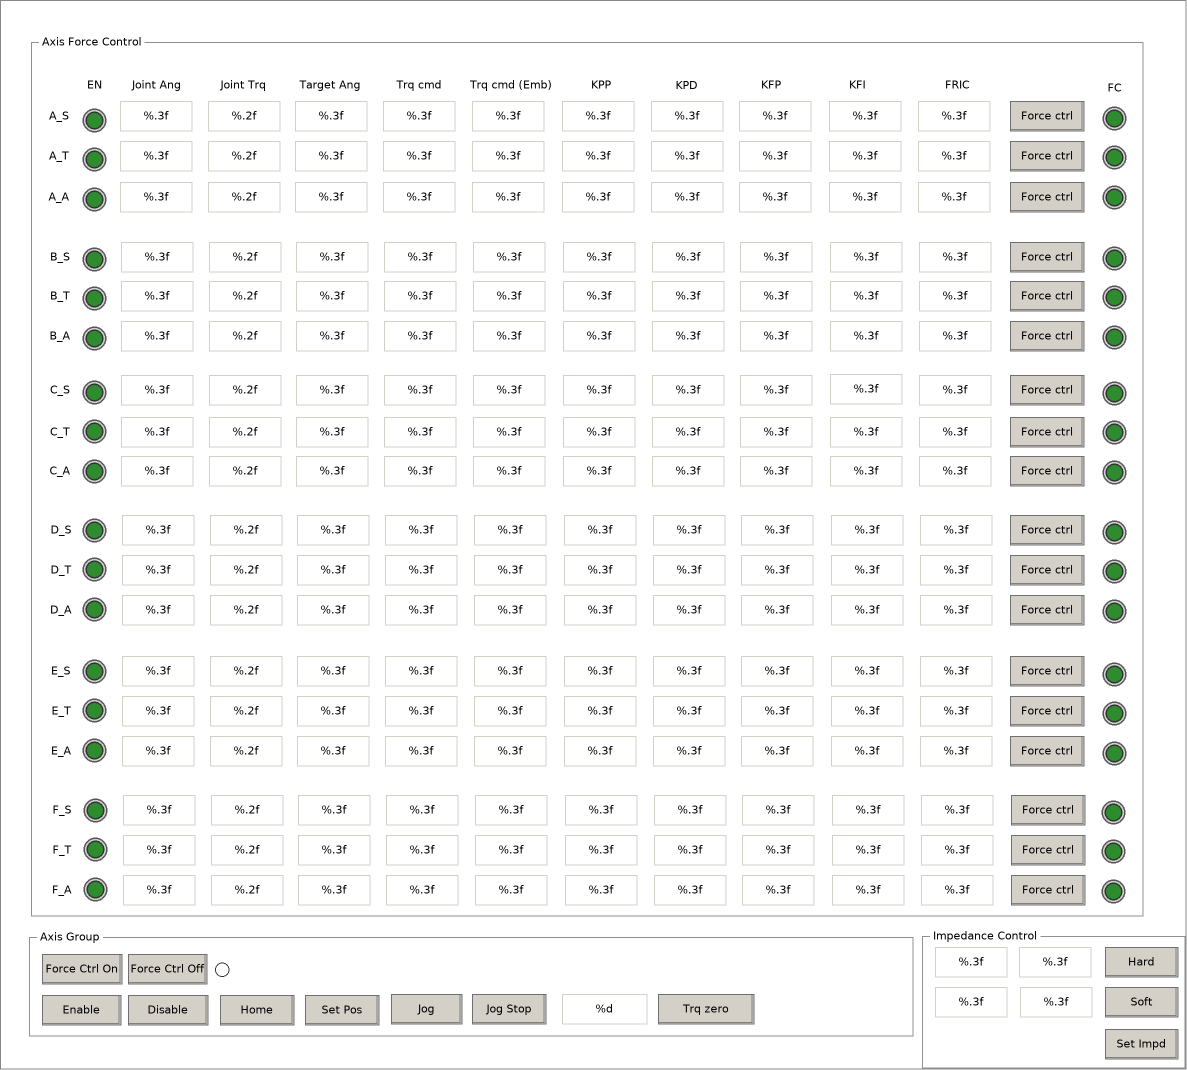
VISUALIZATION ForceControl  // 1187x1070
    GroupBox (31,34 1112x882), "Axis Force Control"
        Label (90,36 71x30), "Joint Ang"
        Label (179,36 67x30), "Joint Trq"
        Label (263,36 72x30), "Target Ang"
        Label (353,36 70x30), "Trq cmd"
        Label (433,36 94x30), "Trq cmd (Emb)"
        Textfield (89,67 72x30), "%.3f", text variable: GVL.motorDrive[0].motorAngle
        Label (545,39 50x24), "KPP"
        Label (632,36 47x31), "KPD"
        Label (800,36 53x30), "KFI"
        Label (714,36 52x30), "KFP"
        Label (900,36 53x30), "FRIC"
        Label (7,72 42x20), "A_S"
        Label (7,112 42x20), "A_T"
        Label (7,153 42x20), "A_A"
        Label (8,213 42x20), "B_S"
        Label (8,252 42x20), "B_T"
        Label (8,292 42x20), "B_A"
        Label (8,346 42x20), "C_S"
        Label (8,388 42x20), "C_T"
        Label (8,427 42x20), "C_A"
        Label (9,486 42x20), "D_S"
        Label (9,526 42x20), "D_T"
        Label (9,566 42x20), "D_A"
        Textfield (89,107 72x30), "%.3f", text variable: GVL.motorDrive[1].motorAngle
        Textfield (89,148 72x30), "%.3f", text variable: GVL.motorDrive[2].motorAngle
        Textfield (90,208 72x30), "%.3f", text variable: GVL.motorDrive[3].motorAngle
        Textfield (90,247 72x30), "%.3f", text variable: GVL.motorDrive[4].motorAngle
        Textfield (90,287 72x30), "%.3f", text variable: GVL.motorDrive[5].motorAngle
        Textfield (91,481 72x30), "%.3f", text variable: GVL.motorDrive[9].motorAngle
        Textfield (177,67 72x30), "%.2f", text variable: GVL.motorDrive[0].trqCalibrated
        Textfield (264,67 72x30), "%.3f", text variable: GVL.motorDrive[0].tgtAngle
            OnMouseClick: write the text variable via Default
        Textfield (352,67 72x30), "%.3f", text variable: GVL.motorDrive[0].trqOutput
        Button (979,67 74x30), "Force ctrl"
            toggle GVL.axisForceCtrlButton[0]
        Button (979,107 74x30), "Force ctrl"
            toggle GVL.axisForceCtrlButton[1]
        Button (979,148 74x30), "Force ctrl"
            toggle GVL.axisForceCtrlButton[2]
        Button (979,208 74x30), "Force ctrl"
            toggle GVL.axisForceCtrlButton[3]
        Button (979,247 74x30), "Force ctrl"
            toggle GVL.axisForceCtrlButton[4]
        Button (979,287 74x30), "Force ctrl"
            toggle GVL.axisForceCtrlButton[5]
        Button (979,341 74x30), "Force ctrl"
            toggle GVL.axisForceCtrlButton[6]
        Button (979,383 74x30), "Force ctrl"
            toggle GVL.axisForceCtrlButton[7]
        Button (979,422 74x30), "Force ctrl"
            toggle GVL.axisForceCtrlButton[8]
        Button (979,481 74x30), "Force ctrl"
            toggle GVL.axisForceCtrlButton[9]
        Button (979,521 74x30), "Force ctrl"
            toggle GVL.axisForceCtrlButton[10]
        Button (979,561 74x30), "Force ctrl"
            toggle GVL.axisForceCtrlButton[11]
        Textfield (620,67 72x30), "%.3f", text variable: GVL.motorDrive[0].bVirtual
            OnMouseClick: write the text variable via Default
        Textfield (708,67 72x30), "%.3f", text variable: GVL.motorDrive[0].kpTrqLoop
            OnMouseClick: write the text variable via Default
        Textfield (798,67 72x30), "%.3f", text variable: GVL.motorDrive[0].kiTrqLoop
            OnMouseClick: write the text variable via Default
        Textfield (887,67 72x30), "%.3f", text variable: GVL.motorDrive[0].reducerColbConstant
            OnMouseClick: write the text variable via Default
        Lamp1 (1070,70 27x29), variable: GVL.axisForceCtrlModeInd[0], style: Lamp-Lamp1-Green
        Label (1057,39 53x30), "FC"
        Label (33,41 61x20), "EN"
        Label (9,627 42x20), "E_S"
        Label (10,766 42x20), "F_S"
        Lamp1 (1070,626 27x29), variable: GVL.axisForceCtrlModeInd[12], style: Lamp-Lamp1-Green
        Lamp1 (1069,764 27x29), variable: GVL.axisForceCtrlModeInd[15], style: Lamp-Lamp1-Green
        Lamp1 (1069,803 27x29), variable: GVL.axisForceCtrlModeInd[16], style: Lamp-Lamp1-Green
        Lamp1 (1069,843 27x29), variable: GVL.axisForceCtrlModeInd[17], style: Lamp-Lamp1-Green
    Textfield (121,375 72x30), "%.3f", text variable: GVL.motorDrive[6].motorAngle
    Textfield (121,417 72x30), "%.3f", text variable: GVL.motorDrive[7].motorAngle
    Textfield (121,456 72x30), "%.3f", text variable: GVL.motorDrive[8].motorAngle
    Textfield (122,555 72x30), "%.3f", text variable: GVL.motorDrive[10].motorAngle
    Textfield (122,595 72x30), "%.3f", text variable: GVL.motorDrive[11].motorAngle
    Textfield (208,141 72x30), "%.2f", text variable: GVL.motorDrive[1].trqCalibrated
    Textfield (208,182 72x30), "%.2f", text variable: GVL.motorDrive[2].trqCalibrated
    Textfield (209,242 72x30), "%.2f", text variable: GVL.motorDrive[3].trqCalibrated
    Textfield (209,281 72x30), "%.2f", text variable: GVL.motorDrive[4].trqCalibrated
    Textfield (209,321 72x30), "%.2f", text variable: GVL.motorDrive[5].trqCalibrated
    Textfield (210,515 72x30), "%.2f", text variable: GVL.motorDrive[9].trqCalibrated
    Textfield (209,375 72x30), "%.2f", text variable: GVL.motorDrive[6].trqCalibrated
    Textfield (209,417 72x30), "%.2f", text variable: GVL.motorDrive[7].trqCalibrated
    Textfield (209,456 72x30), "%.2f", text variable: GVL.motorDrive[8].trqCalibrated
    Textfield (210,555 72x30), "%.2f", text variable: GVL.motorDrive[10].trqCalibrated
    Textfield (210,595 72x30), "%.2f", text variable: GVL.motorDrive[11].trqCalibrated
    Textfield (295,141 72x30), "%.3f", text variable: GVL.motorDrive[1].tgtAngle
        OnMouseClick: write the text variable via Default
    Textfield (295,182 72x30), "%.3f", text variable: GVL.motorDrive[2].tgtAngle
        OnMouseClick: write the text variable via Default
    Textfield (296,242 72x30), "%.3f", text variable: GVL.motorDrive[3].tgtAngle
        OnMouseClick: write the text variable via Default
    Textfield (296,281 72x30), "%.3f", text variable: GVL.motorDrive[4].tgtAngle
        OnMouseClick: write the text variable via Default
    Textfield (296,321 72x30), "%.3f", text variable: GVL.motorDrive[5].tgtAngle
        OnMouseClick: write the text variable via Default
    Textfield (297,515 72x30), "%.3f", text variable: GVL.motorDrive[9].tgtAngle
        OnMouseClick: write the text variable via Default
    Textfield (296,375 72x30), "%.3f", text variable: GVL.motorDrive[6].tgtAngle
        OnMouseClick: write the text variable via Default
    Textfield (296,417 72x30), "%.3f", text variable: GVL.motorDrive[7].tgtAngle
        OnMouseClick: write the text variable via Default
    Textfield (296,456 72x30), "%.3f", text variable: GVL.motorDrive[8].tgtAngle
        OnMouseClick: write the text variable via Default
    Textfield (297,555 72x30), "%.3f", text variable: GVL.motorDrive[10].tgtAngle
        OnMouseClick: write the text variable via Default
    Textfield (297,595 72x30), "%.3f", text variable: GVL.motorDrive[11].tgtAngle
        OnMouseClick: write the text variable via Default
    Textfield (383,141 72x30), "%.3f", text variable: GVL.motorDrive[1].trqOutput
    Textfield (383,182 72x30), "%.3f", text variable: GVL.motorDrive[2].trqOutput
    Textfield (384,242 72x30), "%.3f", text variable: GVL.motorDrive[3].trqOutput
    Textfield (384,281 72x30), "%.3f", text variable: GVL.motorDrive[4].trqOutput
    Textfield (384,321 72x30), "%.3f", text variable: GVL.motorDrive[5].trqOutput
    Textfield (385,515 72x30), "%.3f", text variable: GVL.motorDrive[9].trqOutput
    Textfield (472,101 72x30), "%.3f", text variable: GVL.trqOutputs[0]
    Textfield (562,101 72x30), "%.3f", text variable: GVL.motorDrive[0].kVirtual
        OnMouseClick: write the text variable via Default
    Textfield (384,375 72x30), "%.3f", text variable: GVL.motorDrive[6].trqOutput
    Textfield (384,417 72x30), "%.3f", text variable: GVL.motorDrive[7].trqOutput
    Textfield (384,456 72x30), "%.3f", text variable: GVL.motorDrive[8].trqOutput
    Textfield (385,555 72x30), "%.3f", text variable: GVL.motorDrive[10].trqOutput
    Textfield (385,595 72x30), "%.3f", text variable: GVL.motorDrive[11].trqOutput
    Textfield (472,141 72x30), "%.3f", text variable: GVL.trqOutputs[1]
    Textfield (472,182 72x30), "%.3f", text variable: GVL.trqOutputs[2]
    Textfield (473,242 72x30), "%.3f", text variable: GVL.trqOutputs[3]
    Textfield (473,281 72x30), "%.3f", text variable: GVL.trqOutputs[4]
    Textfield (473,321 72x30), "%.3f", text variable: GVL.trqOutputs[5]
    Textfield (474,515 72x30), "%.3f", text variable: GVL.trqOutputs[9]
    Textfield (473,375 72x30), "%.3f", text variable: GVL.trqOutputs[6]
    Textfield (473,417 72x30), "%.3f", text variable: GVL.trqOutputs[7]
    Textfield (473,456 72x30), "%.3f", text variable: GVL.trqOutputs[8]
    Textfield (474,555 72x30), "%.3f", text variable: GVL.trqOutputs[10]
    Textfield (474,595 72x30), "%.3f", text variable: GVL.trqOutputs[11]
    Textfield (562,141 72x30), "%.3f", text variable: GVL.motorDrive[1].kVirtual
        OnMouseClick: write the text variable via Default
    Textfield (562,182 72x30), "%.3f", text variable: GVL.motorDrive[2].kVirtual
        OnMouseClick: write the text variable via Default
    Textfield (563,242 72x30), "%.3f", text variable: GVL.motorDrive[3].kVirtual
        OnMouseClick: write the text variable via Default
    Textfield (563,281 72x30), "%.3f", text variable: GVL.motorDrive[4].kVirtual
        OnMouseClick: write the text variable via Default
    Textfield (563,321 72x30), "%.3f", text variable: GVL.motorDrive[5].kVirtual
        OnMouseClick: write the text variable via Default
    Textfield (564,515 72x30), "%.3f", text variable: GVL.motorDrive[9].kVirtual
        OnMouseClick: write the text variable via Default
    Textfield (563,375 72x30), "%.3f", text variable: GVL.motorDrive[6].kVirtual
        OnMouseClick: write the text variable via Default
    Textfield (563,417 72x30), "%.3f", text variable: GVL.motorDrive[7].kVirtual
        OnMouseClick: write the text variable via Default
    Textfield (563,456 72x30), "%.3f", text variable: GVL.motorDrive[8].kVirtual
        OnMouseClick: write the text variable via Default
    Textfield (564,555 72x30), "%.3f", text variable: GVL.motorDrive[10].kVirtual
        OnMouseClick: write the text variable via Default
    Textfield (564,595 72x30), "%.3f", text variable: GVL.motorDrive[11].kVirtual
        OnMouseClick: write the text variable via Default
    Textfield (651,141 72x30), "%.3f", text variable: GVL.motorDrive[1].bVirtual
        OnMouseClick: write the text variable via Default
    Textfield (651,182 72x30), "%.3f", text variable: GVL.motorDrive[2].bVirtual
        OnMouseClick: write the text variable via Default
    Textfield (652,242 72x30), "%.3f", text variable: GVL.motorDrive[3].bVirtual
        OnMouseClick: write the text variable via Default
    Textfield (652,281 72x30), "%.3f", text variable: GVL.motorDrive[4].bVirtual
        OnMouseClick: write the text variable via Default
    Textfield (652,321 72x30), "%.3f", text variable: GVL.motorDrive[5].bVirtual
        OnMouseClick: write the text variable via Default
    Textfield (653,515 72x30), "%.3f", text variable: GVL.motorDrive[9].bVirtual
        OnMouseClick: write the text variable via Default
    Textfield (652,375 72x30), "%.3f", text variable: GVL.motorDrive[6].bVirtual
        OnMouseClick: write the text variable via Default
    Textfield (652,417 72x30), "%.3f", text variable: GVL.motorDrive[7].bVirtual
        OnMouseClick: write the text variable via Default
    Textfield (652,456 72x30), "%.3f", text variable: GVL.motorDrive[8].bVirtual
        OnMouseClick: write the text variable via Default
    Textfield (653,555 72x30), "%.3f", text variable: GVL.motorDrive[10].bVirtual
        OnMouseClick: write the text variable via Default
    Textfield (653,595 72x30), "%.3f", text variable: GVL.motorDrive[11].bVirtual
        OnMouseClick: write the text variable via Default
    Textfield (739,141 72x30), "%.3f", text variable: GVL.motorDrive[1].kpTrqLoop
        OnMouseClick: write the text variable via Default
    Textfield (739,182 72x30), "%.3f", text variable: GVL.motorDrive[2].kpTrqLoop
        OnMouseClick: write the text variable via Default
    Textfield (740,242 72x30), "%.3f", text variable: GVL.motorDrive[3].kpTrqLoop
        OnMouseClick: write the text variable via Default
    Textfield (740,281 72x30), "%.3f", text variable: GVL.motorDrive[4].kpTrqLoop
        OnMouseClick: write the text variable via Default
    Textfield (740,321 72x30), "%.3f", text variable: GVL.motorDrive[5].kpTrqLoop
        OnMouseClick: write the text variable via Default
    Textfield (741,515 72x30), "%.3f", text variable: GVL.motorDrive[9].kpTrqLoop
        OnMouseClick: write the text variable via Default
    Textfield (740,375 72x30), "%.3f", text variable: GVL.motorDrive[6].kpTrqLoop
        OnMouseClick: write the text variable via Default
    Textfield (740,417 72x30), "%.3f", text variable: GVL.motorDrive[7].kpTrqLoop
        OnMouseClick: write the text variable via Default
    Textfield (740,456 72x30), "%.3f", text variable: GVL.motorDrive[8].kpTrqLoop
        OnMouseClick: write the text variable via Default
    Textfield (741,555 72x30), "%.3f", text variable: GVL.motorDrive[10].kpTrqLoop
        OnMouseClick: write the text variable via Default
    Textfield (741,595 72x30), "%.3f", text variable: GVL.motorDrive[11].kpTrqLoop
        OnMouseClick: write the text variable via Default
    Textfield (829,141 72x30), "%.3f", text variable: GVL.motorDrive[1].kiTrqLoop
        OnMouseClick: write the text variable via Default
    Textfield (829,182 72x30), "%.3f", text variable: GVL.motorDrive[2].kiTrqLoop
        OnMouseClick: write the text variable via Default
    Textfield (830,242 72x30), "%.3f", text variable: GVL.motorDrive[3].kiTrqLoop
        OnMouseClick: write the text variable via Default
    Textfield (830,281 72x30), "%.3f", text variable: GVL.motorDrive[4].kiTrqLoop
        OnMouseClick: write the text variable via Default
    Textfield (830,321 72x30), "%.3f", text variable: GVL.motorDrive[5].kiTrqLoop
        OnMouseClick: write the text variable via Default
    Textfield (831,515 72x30), "%.3f", text variable: GVL.motorDrive[9].kiTrqLoop
        OnMouseClick: write the text variable via Default
    Textfield (830,374 72x30), "%.3f", text variable: GVL.motorDrive[6].kiTrqLoop
        OnMouseClick: write the text variable via Default
    Textfield (830,417 72x30), "%.3f", text variable: GVL.motorDrive[7].kiTrqLoop
        OnMouseClick: write the text variable via Default
    Textfield (830,456 72x30), "%.3f", text variable: GVL.motorDrive[8].kiTrqLoop
        OnMouseClick: write the text variable via Default
    Textfield (831,555 72x30), "%.3f", text variable: GVL.motorDrive[10].kiTrqLoop
        OnMouseClick: write the text variable via Default
    Textfield (831,595 72x30), "%.3f", text variable: GVL.motorDrive[11].kiTrqLoop
        OnMouseClick: write the text variable via Default
    Textfield (918,141 72x30), "%.3f", text variable: GVL.motorDrive[1].reducerColbConstant
        OnMouseClick: write the text variable via Default
    Textfield (918,182 72x30), "%.3f", text variable: GVL.motorDrive[2].reducerColbConstant
        OnMouseClick: write the text variable via Default
    Textfield (919,242 72x30), "%.3f", text variable: GVL.motorDrive[3].reducerColbConstant
        OnMouseClick: write the text variable via Default
    Textfield (919,281 72x30), "%.3f", text variable: GVL.motorDrive[4].reducerColbConstant
        OnMouseClick: write the text variable via Default
    Textfield (919,321 72x30), "%.3f", text variable: GVL.motorDrive[5].reducerColbConstant
        OnMouseClick: write the text variable via Default
    Textfield (920,515 72x30), "%.3f", text variable: GVL.motorDrive[9].reducerColbConstant
        OnMouseClick: write the text variable via Default
    Textfield (919,375 72x30), "%.3f", text variable: GVL.motorDrive[6].reducerColbConstant
        OnMouseClick: write the text variable via Default
    Textfield (919,417 72x30), "%.3f", text variable: GVL.motorDrive[7].reducerColbConstant
        OnMouseClick: write the text variable via Default
    Textfield (919,456 72x30), "%.3f", text variable: GVL.motorDrive[8].reducerColbConstant
        OnMouseClick: write the text variable via Default
    Textfield (920,555 72x30), "%.3f", text variable: GVL.motorDrive[10].reducerColbConstant
        OnMouseClick: write the text variable via Default
    Textfield (920,595 72x30), "%.3f", text variable: GVL.motorDrive[11].reducerColbConstant
        OnMouseClick: write the text variable via Default
    Lamp1 (1101,143 27x29), variable: GVL.axisForceCtrlModeInd[1], style: Lamp-Lamp1-Green
    Lamp1 (1101,183 27x29), variable: GVL.axisForceCtrlModeInd[2], style: Lamp-Lamp1-Green
    Lamp1 (1101,244 27x29), variable: GVL.axisForceCtrlModeInd[3], style: Lamp-Lamp1-Green
    Lamp1 (1101,379 27x29), variable: GVL.axisForceCtrlModeInd[6], style: Lamp-Lamp1-Green
    Lamp1 (1101,283 27x29), variable: GVL.axisForceCtrlModeInd[4], style: Lamp-Lamp1-Green
    Lamp1 (1101,323 27x29), variable: GVL.axisForceCtrlModeInd[5], style: Lamp-Lamp1-Green
    Lamp1 (1101,418 27x29), variable: GVL.axisForceCtrlModeInd[7], style: Lamp-Lamp1-Green
    Lamp1 (1101,458 27x29), variable: GVL.axisForceCtrlModeInd[8], style: Lamp-Lamp1-Green
    Lamp1 (1101,518 27x29), variable: GVL.axisForceCtrlModeInd[9], style: Lamp-Lamp1-Green
    Lamp1 (1101,557 27x29), variable: GVL.axisForceCtrlModeInd[10], style: Lamp-Lamp1-Green
    Lamp1 (1101,597 27x29), variable: GVL.axisForceCtrlModeInd[11], style: Lamp-Lamp1-Green
    Lamp1 (81,106 27x29), variable: GVL.motorDrive[0].enableBit, style: Lamp-Lamp1-Green
    Lamp1 (81,145 27x29), variable: GVL.motorDrive[1].enableBit, style: Lamp-Lamp1-Green
    Lamp1 (81,185 27x29), variable: GVL.motorDrive[2].enableBit, style: Lamp-Lamp1-Green
    Lamp1 (81,245 27x29), variable: GVL.motorDrive[3].enableBit, style: Lamp-Lamp1-Green
    Lamp1 (81,378 27x29), variable: GVL.motorDrive[6].enableBit, style: Lamp-Lamp1-Green
    Lamp1 (81,284 27x29), variable: GVL.motorDrive[4].enableBit, style: Lamp-Lamp1-Green
    Lamp1 (81,324 27x29), variable: GVL.motorDrive[5].enableBit, style: Lamp-Lamp1-Green
    Lamp1 (81,417 27x29), variable: GVL.motorDrive[7].enableBit, style: Lamp-Lamp1-Green
    Lamp1 (81,457 27x29), variable: GVL.motorDrive[8].enableBit, style: Lamp-Lamp1-Green
    Lamp1 (81,516 27x29), variable: GVL.motorDrive[9].enableBit, style: Lamp-Lamp1-Green
    Lamp1 (81,555 27x29), variable: GVL.motorDrive[10].enableBit, style: Lamp-Lamp1-Green
    Lamp1 (81,595 27x29), variable: GVL.motorDrive[11].enableBit, style: Lamp-Lamp1-Green
    GroupBox (29,929 884x107), "Axis Group"
        Button (13,25 80x30), "Force Ctrl On"
            toggle GVL.forceCtrlGroupButton
        RadioButton (184,26 692x29), variable: GVL.groupSelector
            Areas[1]: Text=Shank
            Areas[2]: Text=Thigh
            Areas[3]: Text=Side
            Areas[4]: Text=LegA
            Areas[5]: Text=LegB
            Areas[6]: Text=LegC
            Areas[7]: Text=LegD
            Areas[8]: Text=LegE
            Areas[9]: Text=LegF
        Button (629,65 96x30), "Trq zero"
            toggle GVL.setTSRZeroButton
        Button (99,25 79x30), "Force Ctrl Off"
            toggle GVL.forceCtrlGroupOffButton
        Button (99,66 80x30), "Disable"
            toggle GVL.disableGroupButton
        Button (13,66 79x30), "Enable"
            toggle GVL.enableGroupButton
        Button (191,66 74x30), "Home"
            toggle GVL.homeGroupButton
        Button (276,66 74x30), "Set Pos"
            toggle GVL.setPosGroupButton
        Button (362,65 71x30), "Jog"
            toggle GVL.jogGroupButton
        Textfield (533,65 85x30), "%d", text variable: GVL.jogGroupVelocity
            OnMouseClick: write the text variable via Default
        Button (443,65 74x30), "Jog Stop"
            toggle GVL.jogStopGroupButton
    GroupBox (922,928 263x140), "Impedance Control"
        Textfield (13,19 72x30), "%.3f", text variable: GVL.kpGroup
            OnMouseClick: write the text variable via Default
        Textfield (97,19 72x30), "%.3f", text variable: GVL.kdGroup
            OnMouseClick: write the text variable via Default
        Textfield (98,59 72x30), "%.3f", text variable: GVL.kiTrqGroup
            OnMouseClick: write the text variable via Default
        Textfield (13,59 72x30), "%.3f", text variable: GVL.kpTrqGroup
            OnMouseClick: write the text variable via Default
        Button (183,19 73x30), "Hard"
            toggle GVL.useHardImpedButton
        Button (183,59 73x30), "Soft"
            toggle GVL.useSoftImpedButton
        Button (183,101 73x30), "Set Impd"
            toggle GVL.setGroupImpedButton
    Label (40,701 42x20), "E_T"
    Label (40,741 42x20), "E_A"
    Textfield (122,656 72x30), "%.3f", text variable: GVL.motorDrive[12].motorAngle
    Button (1010,656 74x30), "Force ctrl"
        toggle GVL.axisForceCtrlButton[12]
    Button (1010,696 74x30), "Force ctrl"
        toggle GVL.axisForceCtrlButton[13]
    Button (1010,736 74x30), "Force ctrl"
        toggle GVL.axisForceCtrlButton[14]
    Textfield (122,696 72x30), "%.3f", text variable: GVL.motorDrive[13].motorAngle
    Textfield (122,736 72x30), "%.3f", text variable: GVL.motorDrive[14].motorAngle
    Textfield (210,656 72x30), "%.2f", text variable: GVL.motorDrive[12].trqCalibrated
    Textfield (210,696 72x30), "%.2f", text variable: GVL.motorDrive[13].trqCalibrated
    Textfield (210,736 72x30), "%.2f", text variable: GVL.motorDrive[14].trqCalibrated
    Textfield (297,656 72x30), "%.3f", text variable: GVL.motorDrive[12].tgtAngle
        OnMouseClick: write the text variable via Default
    Textfield (297,696 72x30), "%.3f", text variable: GVL.motorDrive[13].tgtAngle
        OnMouseClick: write the text variable via Default
    Textfield (297,736 72x30), "%.3f", text variable: GVL.motorDrive[14].tgtAngle
        OnMouseClick: write the text variable via Default
    Textfield (385,656 72x30), "%.3f", text variable: GVL.motorDrive[12].trqOutput
    Textfield (385,696 72x30), "%.3f", text variable: GVL.motorDrive[13].trqOutput
    Textfield (385,736 72x30), "%.3f", text variable: GVL.motorDrive[14].trqOutput
    Textfield (474,656 72x30), "%.3f", text variable: GVL.trqOutputs[12]
    Textfield (474,696 72x30), "%.3f", text variable: GVL.trqOutputs[13]
    Textfield (474,736 72x30), "%.3f", text variable: GVL.trqOutputs[14]
    Textfield (564,656 72x30), "%.3f", text variable: GVL.motorDrive[12].kVirtual
        OnMouseClick: write the text variable via Default
    Textfield (564,696 72x30), "%.3f", text variable: GVL.motorDrive[13].kVirtual
        OnMouseClick: write the text variable via Default
    Textfield (564,736 72x30), "%.3f", text variable: GVL.motorDrive[14].kVirtual
        OnMouseClick: write the text variable via Default
    Textfield (653,656 72x30), "%.3f", text variable: GVL.motorDrive[12].bVirtual
        OnMouseClick: write the text variable via Default
    Textfield (653,696 72x30), "%.3f", text variable: GVL.motorDrive[13].bVirtual
        OnMouseClick: write the text variable via Default
    Textfield (653,736 72x30), "%.3f", text variable: GVL.motorDrive[14].bVirtual
        OnMouseClick: write the text variable via Default
    Textfield (741,656 72x30), "%.3f", text variable: GVL.motorDrive[12].kpTrqLoop
        OnMouseClick: write the text variable via Default
    Textfield (741,696 72x30), "%.3f", text variable: GVL.motorDrive[13].kpTrqLoop
        OnMouseClick: write the text variable via Default
    Textfield (741,736 72x30), "%.3f", text variable: GVL.motorDrive[14].kpTrqLoop
        OnMouseClick: write the text variable via Default
    Textfield (831,656 72x30), "%.3f", text variable: GVL.motorDrive[12].kiTrqLoop
        OnMouseClick: write the text variable via Default
    Textfield (831,696 72x30), "%.3f", text variable: GVL.motorDrive[13].kiTrqLoop
        OnMouseClick: write the text variable via Default
    Textfield (831,736 72x30), "%.3f", text variable: GVL.motorDrive[14].kiTrqLoop
        OnMouseClick: write the text variable via Default
    Textfield (920,656 72x30), "%.3f", text variable: GVL.motorDrive[12].reducerColbConstant
        OnMouseClick: write the text variable via Default
    Textfield (920,696 72x30), "%.3f", text variable: GVL.motorDrive[13].reducerColbConstant
        OnMouseClick: write the text variable via Default
    Textfield (920,736 72x30), "%.3f", text variable: GVL.motorDrive[14].reducerColbConstant
        OnMouseClick: write the text variable via Default
    Lamp1 (81,657 27x29), variable: GVL.motorDrive[12].enableBit, style: Lamp-Lamp1-Green
    Lamp1 (81,696 27x29), variable: GVL.motorDrive[13].enableBit, style: Lamp-Lamp1-Green
    Lamp1 (81,736 27x29), variable: GVL.motorDrive[14].enableBit, style: Lamp-Lamp1-Green
    Label (41,840 42x20), "F_T"
    Label (41,880 42x20), "F_A"
    Textfield (123,795 72x30), "%.3f", text variable: GVL.motorDrive[15].motorAngle
    Button (1011,795 74x30), "Force ctrl"
        toggle GVL.axisForceCtrlButton[15]
    Button (1011,835 74x30), "Force ctrl"
        toggle GVL.axisForceCtrlButton[16]
    Button (1011,875 74x30), "Force ctrl"
        toggle GVL.axisForceCtrlButton[17]
    Textfield (123,835 72x30), "%.3f", text variable: GVL.motorDrive[16].motorAngle
    Textfield (123,875 72x30), "%.3f", text variable: GVL.motorDrive[17].motorAngle
    Textfield (211,795 72x30), "%.2f", text variable: GVL.motorDrive[15].trqCalibrated
    Textfield (211,835 72x30), "%.2f", text variable: GVL.motorDrive[16].trqCalibrated
    Textfield (211,875 72x30), "%.2f", text variable: GVL.motorDrive[17].trqCalibrated
    Textfield (298,795 72x30), "%.3f", text variable: GVL.motorDrive[15].tgtAngle
        OnMouseClick: write the text variable via Default
    Textfield (298,835 72x30), "%.3f", text variable: GVL.motorDrive[16].tgtAngle
        OnMouseClick: write the text variable via Default
    Textfield (298,875 72x30), "%.3f", text variable: GVL.motorDrive[17].tgtAngle
        OnMouseClick: write the text variable via Default
    Textfield (386,795 72x30), "%.3f", text variable: GVL.motorDrive[15].trqOutput
    Textfield (386,835 72x30), "%.3f", text variable: GVL.motorDrive[16].trqOutput
    Textfield (386,875 72x30), "%.3f", text variable: GVL.motorDrive[17].trqOutput
    Textfield (475,795 72x30), "%.3f", text variable: GVL.trqOutputs[15]
    Textfield (475,835 72x30), "%.3f", text variable: GVL.trqOutputs[16]
    Textfield (475,875 72x30), "%.3f", text variable: GVL.trqOutputs[17]
    Textfield (565,795 72x30), "%.3f", text variable: GVL.motorDrive[15].kVirtual
        OnMouseClick: write the text variable via Default
    Textfield (565,835 72x30), "%.3f", text variable: GVL.motorDrive[16].kVirtual
        OnMouseClick: write the text variable via Default
    Textfield (565,875 72x30), "%.3f", text variable: GVL.motorDrive[17].kVirtual
        OnMouseClick: write the text variable via Default
    Textfield (654,795 72x30), "%.3f", text variable: GVL.motorDrive[15].bVirtual
        OnMouseClick: write the text variable via Default
    Textfield (654,835 72x30), "%.3f", text variable: GVL.motorDrive[16].bVirtual
        OnMouseClick: write the text variable via Default
    Textfield (654,875 72x30), "%.3f", text variable: GVL.motorDrive[17].bVirtual
        OnMouseClick: write the text variable via Default
    Textfield (742,795 72x30), "%.3f", text variable: GVL.motorDrive[15].kpTrqLoop
        OnMouseClick: write the text variable via Default
    Textfield (742,835 72x30), "%.3f", text variable: GVL.motorDrive[16].kpTrqLoop
        OnMouseClick: write the text variable via Default
    Textfield (742,875 72x30), "%.3f", text variable: GVL.motorDrive[17].kpTrqLoop
        OnMouseClick: write the text variable via Default
    Textfield (832,795 72x30), "%.3f", text variable: GVL.motorDrive[15].kiTrqLoop
        OnMouseClick: write the text variable via Default
    Textfield (832,835 72x30), "%.3f", text variable: GVL.motorDrive[16].kiTrqLoop
        OnMouseClick: write the text variable via Default
    Textfield (832,875 72x30), "%.3f", text variable: GVL.motorDrive[17].kiTrqLoop
        OnMouseClick: write the text variable via Default
    Textfield (921,795 72x30), "%.3f", text variable: GVL.motorDrive[15].reducerColbConstant
        OnMouseClick: write the text variable via Default
    Textfield (921,835 72x30), "%.3f", text variable: GVL.motorDrive[16].reducerColbConstant
        OnMouseClick: write the text variable via Default
    Textfield (921,875 72x30), "%.3f", text variable: GVL.motorDrive[17].reducerColbConstant
        OnMouseClick: write the text variable via Default
    Lamp1 (82,796 27x29), variable: GVL.motorDrive[15].enableBit, style: Lamp-Lamp1-Green
    Lamp1 (82,835 27x29), variable: GVL.motorDrive[16].enableBit, style: Lamp-Lamp1-Green
    Lamp1 (82,875 27x29), variable: GVL.motorDrive[17].enableBit, style: Lamp-Lamp1-Green
    Lamp1 (1101,699 27x29), variable: GVL.axisForceCtrlModeInd[13], style: Lamp-Lamp1-Green
    Lamp1 (1101,739 27x29), variable: GVL.axisForceCtrlModeInd[14], style: Lamp-Lamp1-Green
END_VISUALIZATION

(* stored: Version 1.1.0.1, ProductVersion 3.1.4024.2
   Visu ForceControl: Id {0c241e3c-c466-4f45-aaaf-7dff6844cb63} *)
